(*
Casts I_Component to I_State
*)
FUNCTION ICompToIState : Result
VAR_INPUT
	iSource	: I_Component;
END_VAR
VAR_OUTPUT
	iDest	: I_State;
END_VAR

IF iSource = 0 THEN
	ICompToIState := Err.Itf0;
	RETURN;
END_IF

IF __QUERYINTERFACE(iSource, iDest) THEN
	ICompToIState := Ok;
ELSE
	iDest := 0;
	ICompToIState := Err.NoMatch;
END_IF

END_FUNCTION

(* stored: Version 1.1.0.1
   POU ICompToIState: Id {4f07989d-6b80-4af7-8c3a-fc64f8e2cb2a}, SpecialFunc None *)
